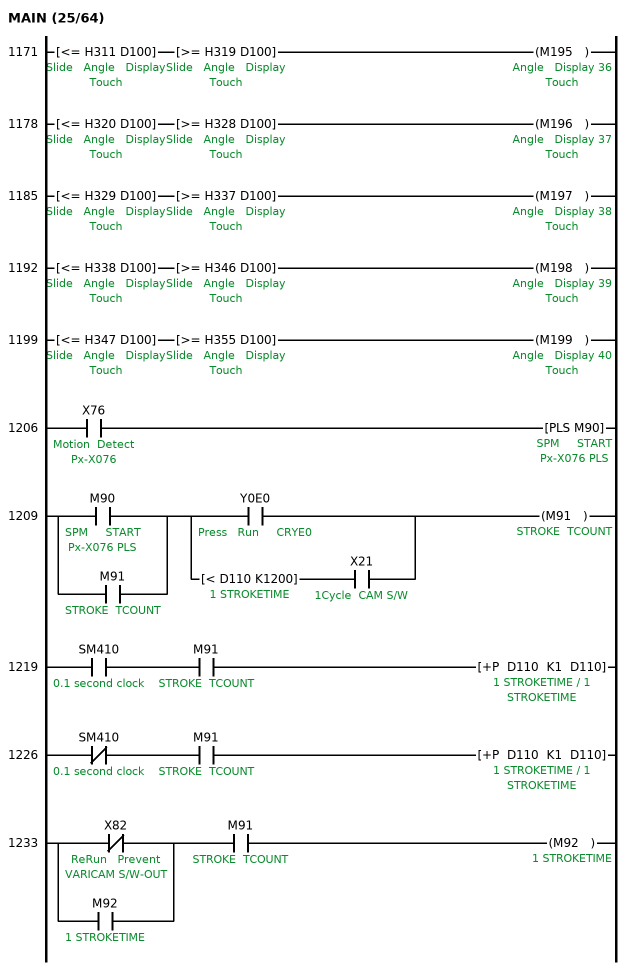
[picture p24: ladder of MAIN, rungs at steps 1171 to 1233]
1171  LD<=    H311 D100  ; Slide   Angle   Display Touch
      AND>=   H319 D100  ; Slide   Angle   Display Touch
      OUT     M195  ; Angle   Display 36      Touch
1178  LD<=    H320 D100  ; Slide   Angle   Display Touch
      AND>=   H328 D100  ; Slide   Angle   Display Touch
      OUT     M196  ; Angle   Display 37      Touch
1185  LD<=    H329 D100  ; Slide   Angle   Display Touch
      AND>=   H337 D100  ; Slide   Angle   Display Touch
      OUT     M197  ; Angle   Display 38      Touch
1192  LD<=    H338 D100  ; Slide   Angle   Display Touch
      AND>=   H346 D100  ; Slide   Angle   Display Touch
      OUT     M198  ; Angle   Display 39      Touch
1199  LD<=    H347 D100  ; Slide   Angle   Display Touch
      AND>=   H355 D100  ; Slide   Angle   Display Touch
      OUT     M199  ; Angle   Display 40      Touch
1206  LD      X76  ; Motion  Detect  Px-X076
      PLS     M90  ; SPM     START   Px-X076 PLS
1209  LD      M90  ; SPM     START   Px-X076 PLS
      OR      M91  ; STROKE  TCOUNT
      LD      Y0E0  ; Press   Run     CRYE0
      LD<     D110 K1200  ; 1 STROKETIME
      AND     X21  ; 1Cycle  CAM S/W
      ORB
      ANB
      OUT     M91  ; STROKE  TCOUNT
1219  LD      SM410  ; 0.1 second clock
      AND     M91  ; STROKE  TCOUNT
      +P      D110 K1 D110
1226  LDI     SM410  ; 0.1 second clock
      AND     M91  ; STROKE  TCOUNT
      +P      D110 K1 D110
1233  LDI     X82  ; ReRun   Prevent VARICAM S/W-OUT
      OR      M92  ; 1 STROKETIME
      AND     M91  ; STROKE  TCOUNT
      OUT     M92  ; 1 STROKETIME
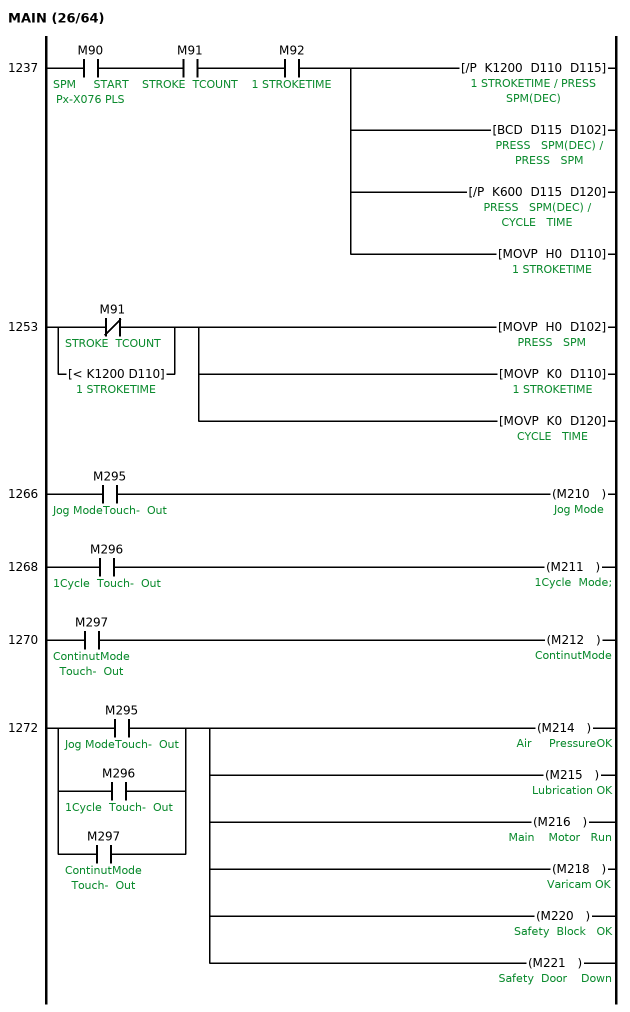
1237  LD      M90  ; SPM     START   Px-X076 PLS
      AND     M91  ; STROKE  TCOUNT
      AND     M92  ; 1 STROKETIME
      /P      K1200 D110 D115  ; PRESS   SPM(DEC)
      BCD     D115 D102  ; PRESS   SPM
      /P      K600 D115 D120  ; CYCLE   TIME
      MOVP    H0 D110
1253  LDI     M91  ; STROKE  TCOUNT
      OR<     K1200 D110  ; 1 STROKETIME
      MOVP    H0 D102
      MOVP    K0 D110
      MOVP    K0 D120
1266  LD      M295  ; Jog ModeTouch-  Out
      OUT     M210  ; Jog Mode
1268  LD      M296  ; 1Cycle  Touch-  Out
      OUT     M211  ; 1Cycle  Mode;
1270  LD      M297  ; ContinutMode    Touch-  Out
      OUT     M212  ; ContinutMode
1272  LD      M295  ; Jog ModeTouch-  Out
      OR      M296  ; 1Cycle  Touch-  Out
      OR      M297  ; ContinutMode    Touch-  Out
      OUT     M214  ; Air     PressureOK
      OUT     M215  ; Lubrication OK
      OUT     M216  ; Main    Motor   Run
      OUT     M218  ; Varicam OK
      OUT     M220  ; Safety  Block   OK
      OUT     M221  ; Safety  Door    Down
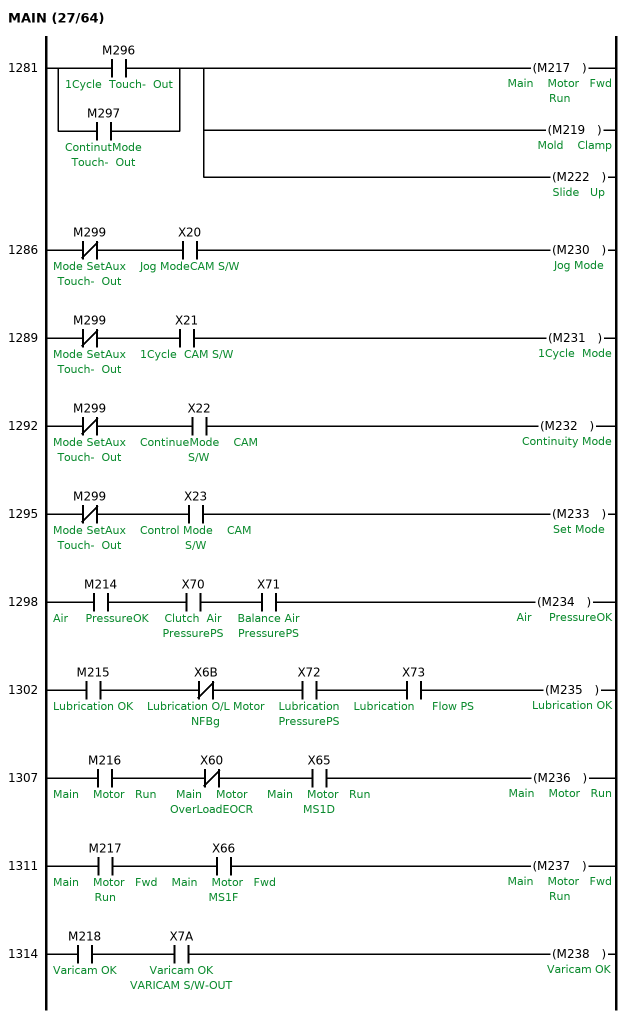
1281  LD      M296  ; 1Cycle  Touch-  Out
      OR      M297  ; ContinutMode    Touch-  Out
      OUT     M217  ; Main    Motor   Fwd Run
      OUT     M219  ; Mold    Clamp
      OUT     M222  ; Slide   Up
1286  LDI     M299  ; Mode SetAux     Touch-  Out
      AND     X20  ; Jog ModeCAM S/W
      OUT     M230  ; Jog Mode
1289  LDI     M299  ; Mode SetAux     Touch-  Out
      AND     X21  ; 1Cycle  CAM S/W
      OUT     M231  ; 1Cycle  Mode
1292  LDI     M299  ; Mode SetAux     Touch-  Out
      AND     X22  ; ContinueMode    CAM S/W
      OUT     M232  ; Continuity Mode
1295  LDI     M299  ; Mode SetAux     Touch-  Out
      AND     X23  ; Control Mode    CAM S/W
      OUT     M233  ; Set Mode
1298  LD      M214  ; Air     PressureOK
      AND     X70  ; Clutch  Air     PressurePS
      AND     X71  ; Balance Air     PressurePS
      OUT     M234  ; Air     PressureOK
1302  LD      M215  ; Lubrication OK
      ANI     X6B  ; Lubrication O/L Motor   NFBg
      AND     X72  ; Lubrication     PressurePS
      AND     X73  ; Lubrication     Flow PS
      OUT     M235  ; Lubrication OK
1307  LD      M216  ; Main    Motor   Run
      ANI     X60  ; Main    Motor   OverLoadEOCR
      AND     X65  ; Main    Motor   Run MS1D
      OUT     M236  ; Main    Motor   Run
1311  LD      M217  ; Main    Motor   Fwd Run
      AND     X66  ; Main    Motor   Fwd     MS1F
      OUT     M237  ; Main    Motor   Fwd Run
1314  LD      M218  ; Varicam OK
      AND     X7A  ; Varicam OK      VARICAM S/W-OUT
      OUT     M238  ; Varicam OK
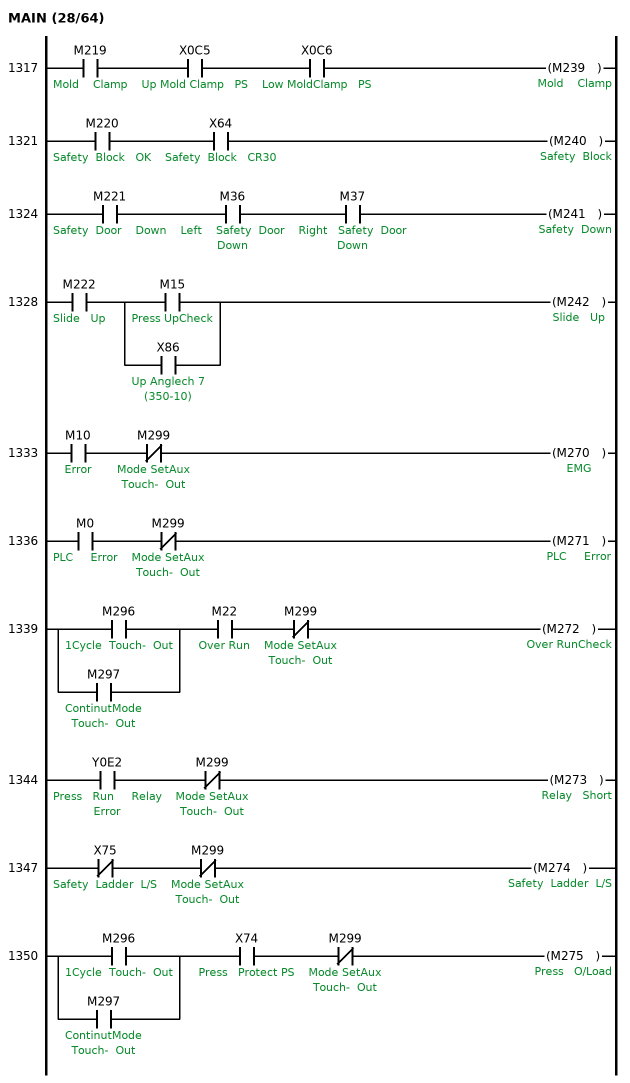
1317  LD      M219  ; Mold    Clamp
      AND     X0C5  ; Up Mold Clamp   PS
      AND     X0C6  ; Low MoldClamp   PS
      OUT     M239  ; Mold    Clamp
1321  LD      M220  ; Safety  Block   OK
      AND     X64  ; Safety  Block   CR30
      OUT     M240  ; Safety  Block
1324  LD      M221  ; Safety  Door    Down
      AND     M36  ; Left    Safety  Door    Down
      AND     M37  ; Right   Safety  Door    Down
      OUT     M241  ; Safety  Down
1328  LD      M222  ; Slide   Up
      LD      M15  ; Press UpCheck
      OR      X86  ; Up Anglech 7    (350-10)
      ANB
      OUT     M242  ; Slide   Up
1333  LD      M10  ; Error
      ANI     M299  ; Mode SetAux     Touch-  Out
      OUT     M270  ; EMG
1336  LD      M0  ; PLC     Error
      ANI     M299  ; Mode SetAux     Touch-  Out
      OUT     M271  ; PLC     Error
1339  LD      M296  ; 1Cycle  Touch-  Out
      OR      M297  ; ContinutMode    Touch-  Out
      AND     M22  ; Over Run
      ANI     M299  ; Mode SetAux     Touch-  Out
      OUT     M272  ; Over RunCheck
1344  LD      Y0E2  ; Press   Run     Relay   Error
      ANI     M299  ; Mode SetAux     Touch-  Out
      OUT     M273  ; Relay   Short
1347  LDI     X75  ; Safety  Ladder  L/S
      ANI     M299  ; Mode SetAux     Touch-  Out
      OUT     M274  ; Safety  Ladder  L/S
1350  LD      M296  ; 1Cycle  Touch-  Out
      OR      M297  ; ContinutMode    Touch-  Out
      AND     X74  ; Press   Protect PS
      ANI     M299  ; Mode SetAux     Touch-  Out
      OUT     M275  ; Press   O/Load
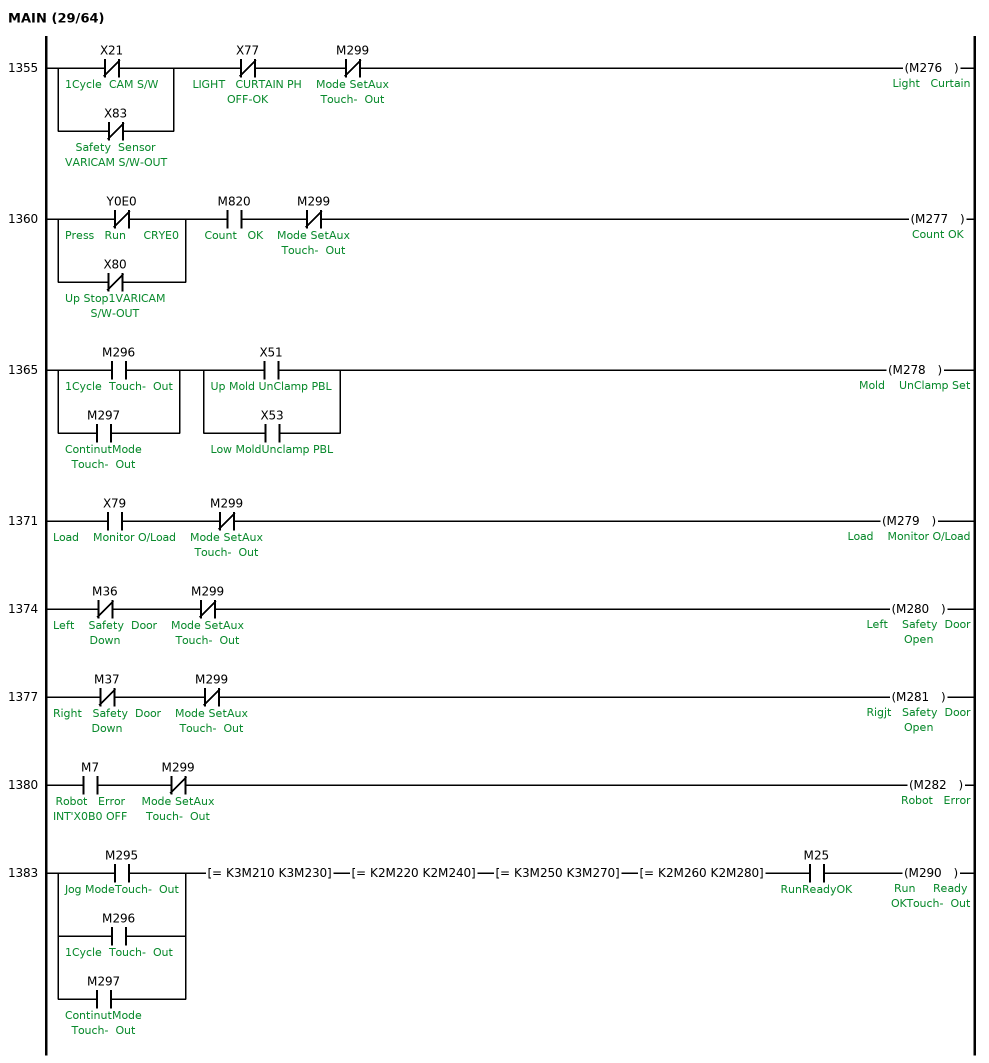
1355  LDI     X21  ; 1Cycle  CAM S/W
      ORI     X83  ; Safety  Sensor  VARICAM S/W-OUT
      ANI     X77  ; LIGHT   CURTAIN PH      OFF-OK
      ANI     M299  ; Mode SetAux     Touch-  Out
      OUT     M276  ; Light   Curtain
1360  LDI     Y0E0  ; Press   Run     CRYE0
      ORI     X80  ; Up Stop1VARICAM S/W-OUT
      AND     M820  ; Count   OK
      ANI     M299  ; Mode SetAux     Touch-  Out
      OUT     M277  ; Count OK
1365  LD      M296  ; 1Cycle  Touch-  Out
      OR      M297  ; ContinutMode    Touch-  Out
      LD      X51  ; Up Mold UnClamp PBL
      OR      X53  ; Low MoldUnclamp PBL
      ANB
      OUT     M278  ; Mold    UnClamp Set
1371  LD      X79  ; Load    Monitor O/Load
      ANI     M299  ; Mode SetAux     Touch-  Out
      OUT     M279  ; Load    Monitor O/Load
1374  LDI     M36  ; Left    Safety  Door    Down
      ANI     M299  ; Mode SetAux     Touch-  Out
      OUT     M280  ; Left    Safety  Door    Open
1377  LDI     M37  ; Right   Safety  Door    Down
      ANI     M299  ; Mode SetAux     Touch-  Out
      OUT     M281  ; Rigjt   Safety  Door    Open
1380  LD      M7  ; Robot   Error   INT'X0B0 OFF
      ANI     M299  ; Mode SetAux     Touch-  Out
      OUT     M282  ; Robot   Error
1383  LD      M295  ; Jog ModeTouch-  Out
      OR      M296  ; 1Cycle  Touch-  Out
      OR      M297  ; ContinutMode    Touch-  Out
      AND=    K3M210 K3M230  ; Jog Mode / Jog Mode
      AND=    K2M220 K2M240  ; Safety  Block   OK / Safety  Block
      AND=    K3M250 K3M270  ; EMG / EMG
      AND=    K2M260 K2M280  ; Left    Safety  Door    Open / Left    Safety  Door    Open
      AND     M25  ; RunReadyOK
      OUT     M290  ; Run     Ready OKTouch-  Out
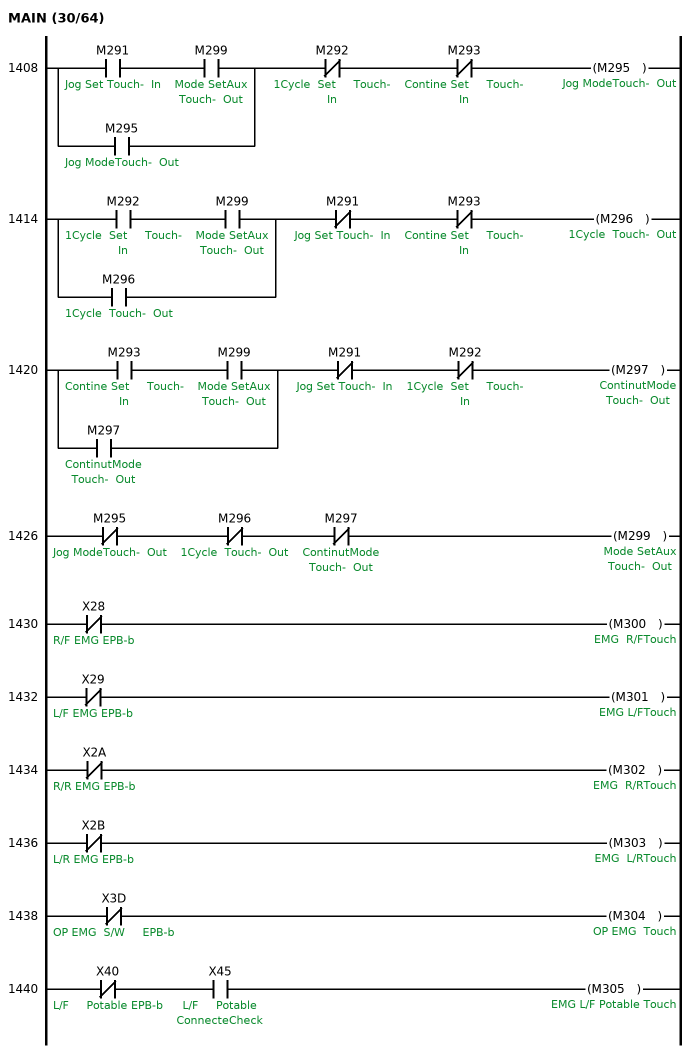
1408  LD      M291  ; Jog Set Touch-  In
      AND     M299  ; Mode SetAux     Touch-  Out
      OR      M295  ; Jog ModeTouch-  Out
      ANI     M292  ; 1Cycle  Set     Touch-  In
      ANI     M293  ; Contine Set     Touch-  In
      OUT     M295  ; Jog ModeTouch-  Out
1414  LD      M292  ; 1Cycle  Set     Touch-  In
      AND     M299  ; Mode SetAux     Touch-  Out
      OR      M296  ; 1Cycle  Touch-  Out
      ANI     M291  ; Jog Set Touch-  In
      ANI     M293  ; Contine Set     Touch-  In
      OUT     M296  ; 1Cycle  Touch-  Out
1420  LD      M293  ; Contine Set     Touch-  In
      AND     M299  ; Mode SetAux     Touch-  Out
      OR      M297  ; ContinutMode    Touch-  Out
      ANI     M291  ; Jog Set Touch-  In
      ANI     M292  ; 1Cycle  Set     Touch-  In
      OUT     M297  ; ContinutMode    Touch-  Out
1426  LDI     M295  ; Jog ModeTouch-  Out
      ANI     M296  ; 1Cycle  Touch-  Out
      ANI     M297  ; ContinutMode    Touch-  Out
      OUT     M299  ; Mode SetAux     Touch-  Out
1430  LDI     X28  ; R/F EMG EPB-b
      OUT     M300  ; EMG  R/FTouch
1432  LDI     X29  ; L/F EMG EPB-b
      OUT     M301  ; EMG L/FTouch
1434  LDI     X2A  ; R/R EMG EPB-b
      OUT     M302  ; EMG  R/RTouch
1436  LDI     X2B  ; L/R EMG EPB-b
      OUT     M303  ; EMG  L/RTouch
1438  LDI     X3D  ; OP EMG  S/W     EPB-b
      OUT     M304  ; OP EMG  Touch
1440  LDI     X40  ; L/F     Potable EPB-b
      AND     X45  ; L/F     Potable ConnecteCheck
      OUT     M305  ; EMG L/F Potable Touch
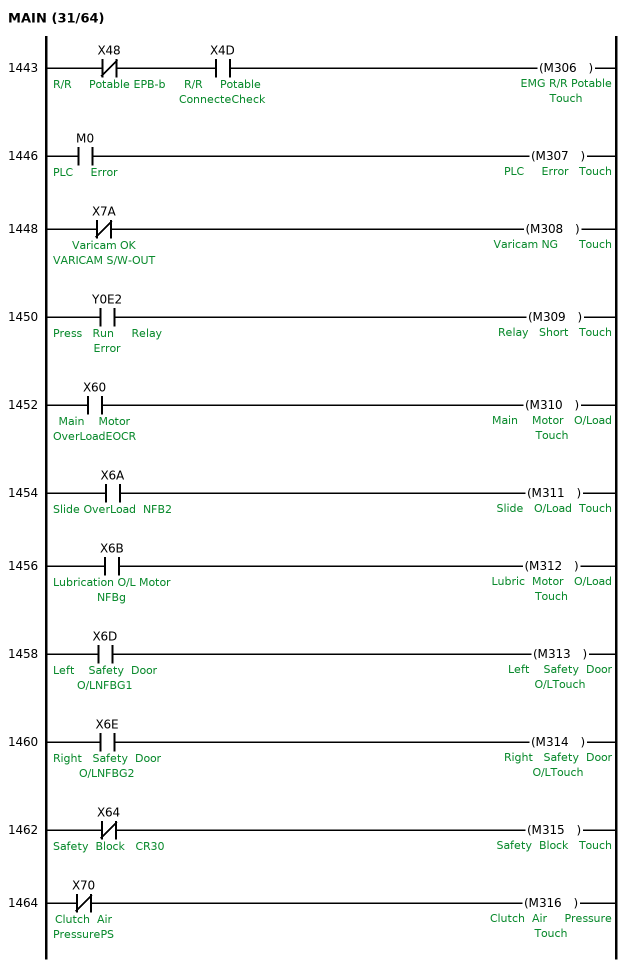
1443  LDI     X48  ; R/R     Potable EPB-b
      AND     X4D  ; R/R     Potable ConnecteCheck
      OUT     M306  ; EMG R/R Potable Touch
1446  LD      M0  ; PLC     Error
      OUT     M307  ; PLC     Error   Touch
1448  LDI     X7A  ; Varicam OK      VARICAM S/W-OUT
      OUT     M308  ; Varicam NG      Touch
1450  LD      Y0E2  ; Press   Run     Relay   Error
      OUT     M309  ; Relay   Short   Touch
1452  LD      X60  ; Main    Motor   OverLoadEOCR
      OUT     M310  ; Main    Motor   O/Load  Touch
1454  LD      X6A  ; Slide OverLoad  NFB2
      OUT     M311  ; Slide   O/Load  Touch
1456  LD      X6B  ; Lubrication O/L Motor   NFBg
      OUT     M312  ; Lubric  Motor   O/Load  Touch
1458  LD      X6D  ; Left    Safety  Door O/LNFBG1
      OUT     M313  ; Left    Safety  Door O/LTouch
1460  LD      X6E  ; Right   Safety  Door O/LNFBG2
      OUT     M314  ; Right   Safety  Door O/LTouch
1462  LDI     X64  ; Safety  Block   CR30
      OUT     M315  ; Safety  Block   Touch
1464  LDI     X70  ; Clutch  Air     PressurePS
      OUT     M316  ; Clutch  Air     Pressure Touch
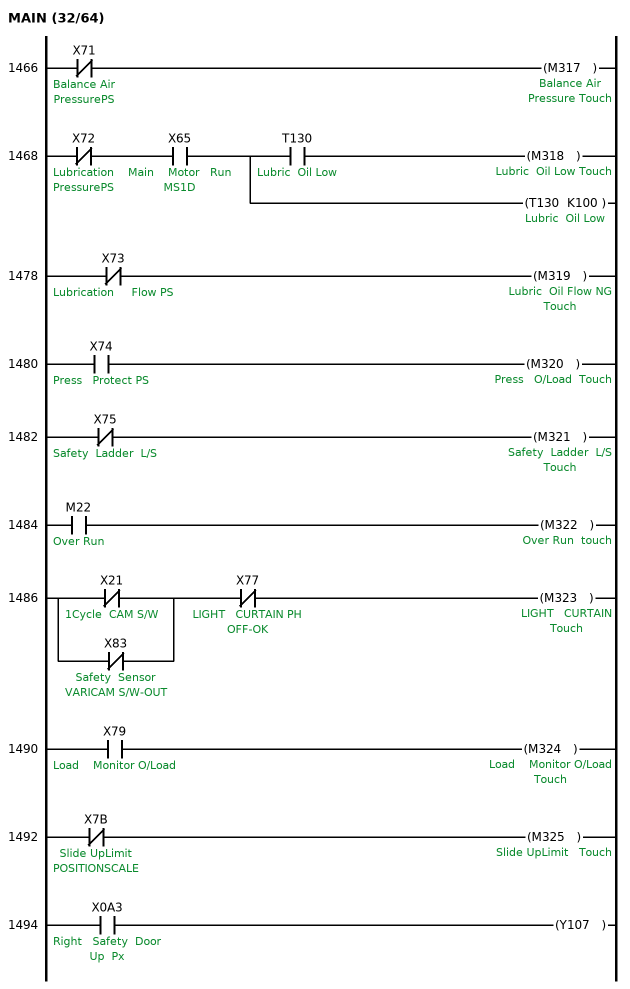
1466  LDI     X71  ; Balance Air     PressurePS
      OUT     M317  ; Balance Air     Pressure Touch
1468  LDI     X72  ; Lubrication     PressurePS
      AND     X65  ; Main    Motor   Run MS1D
      MPS
      AND     T130  ; Lubric  Oil Low
      OUT     M318  ; Lubric  Oil Low Touch
      MPP
      OUT     T130 K100  ; Lubric  Oil Low
1478  LDI     X73  ; Lubrication     Flow PS
      OUT     M319  ; Lubric  Oil Flow NG     Touch
1480  LD      X74  ; Press   Protect PS
      OUT     M320  ; Press   O/Load  Touch
1482  LDI     X75  ; Safety  Ladder  L/S
      OUT     M321  ; Safety  Ladder  L/S     Touch
1484  LD      M22  ; Over Run
      OUT     M322  ; Over Run  touch
1486  LDI     X21  ; 1Cycle  CAM S/W
      ORI     X83  ; Safety  Sensor  VARICAM S/W-OUT
      ANI     X77  ; LIGHT   CURTAIN PH      OFF-OK
      OUT     M323  ; LIGHT   CURTAIN Touch
1490  LD      X79  ; Load    Monitor O/Load
      OUT     M324  ; Load    Monitor O/Load  Touch
1492  LDI     X7B  ; Slide UpLimit   POSITIONSCALE
      OUT     M325  ; Slide UpLimit   Touch
1494  LD      X0A3  ; Right   Safety  Door Up  Px
      OUT     Y107
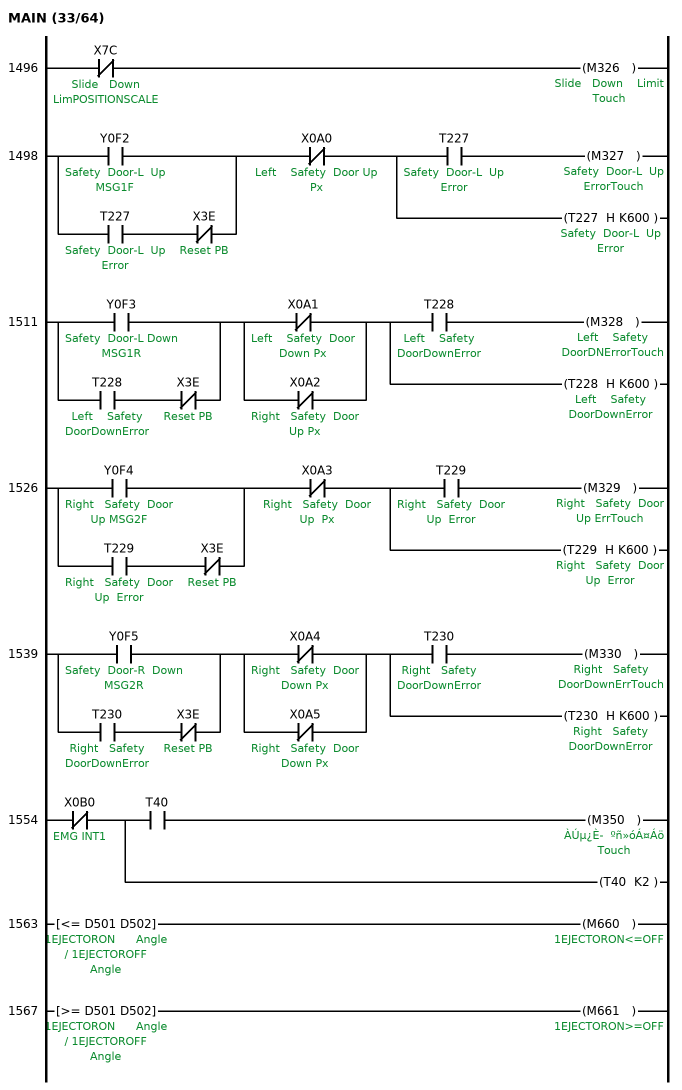
1496  LDI     X7C  ; Slide   Down LimPOSITIONSCALE
      OUT     M326  ; Slide   Down    Limit   Touch
1498  LD      Y0F2  ; Safety  Door-L  Up MSG1F
      LD      T227  ; Safety  Door-L  Up Error
      ANI     X3E  ; Reset PB
      ORB
      ANI     X0A0  ; Left    Safety  Door Up Px
      MPS
      AND     T227  ; Safety  Door-L  Up Error
      OUT     M327  ; Safety  Door-L  Up ErrorTouch
      MPP
      OUTH    T227 K600  ; Safety  Door-L  Up Error
1511  LD      Y0F3  ; Safety  Door-L Down     MSG1R
      LD      T228  ; Left    Safety  DoorDownError
      ANI     X3E  ; Reset PB
      ORB
      LDI     X0A1  ; Left    Safety  Door    Down Px
      ORI     X0A2  ; Right   Safety  Door Up Px
      ANB
      MPS
      AND     T228  ; Left    Safety  DoorDownError
      OUT     M328  ; Left    Safety  DoorDNErrorTouch
      MPP
      OUTH    T228 K600  ; Left    Safety  DoorDownError
1526  LD      Y0F4  ; Right   Safety  Door Up MSG2F
      LD      T229  ; Right   Safety  Door Up  Error
      ANI     X3E  ; Reset PB
      ORB
      ANI     X0A3  ; Right   Safety  Door Up  Px
      MPS
      AND     T229  ; Right   Safety  Door Up  Error
      OUT     M329  ; Right   Safety  Door Up ErrTouch
      MPP
      OUTH    T229 K600  ; Right   Safety  Door Up  Error
1539  LD      Y0F5  ; Safety  Door-R  Down    MSG2R
      LD      T230  ; Right   Safety  DoorDownError
      ANI     X3E  ; Reset PB
      ORB
      LDI     X0A4  ; Right   Safety  Door    Down Px
      ORI     X0A5  ; Right   Safety  Door    Down Px
      ANB
      MPS
      AND     T230  ; Right   Safety  DoorDownError
      OUT     M330  ; Right   Safety  DoorDownErrTouch
      MPP
      OUTH    T230 K600  ; Right   Safety  DoorDownError
1554  LDI     X0B0  ; EMG INT1
      MPS
      AND     T40
      OUT     M350  ; ÀÚµ¿È­  ºñ»óÁ¤ÁöTouch
      MPP
      OUT     T40 K2
1563  LD<=    D501 D502  ; 1EJECTORON      Angle / 1EJECTOROFF     Angle
      OUT     M660  ; 1EJECTORON<=OFF
1567  LD>=    D501 D502  ; 1EJECTORON      Angle / 1EJECTOROFF     Angle
      OUT     M661  ; 1EJECTORON>=OFF
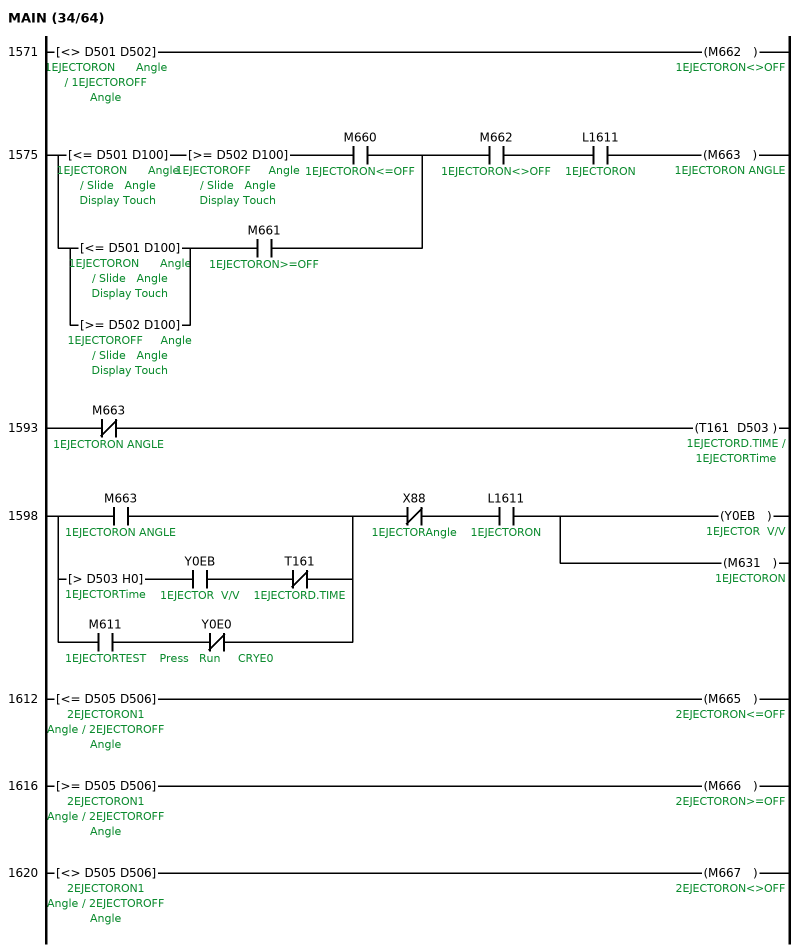
1571  LD<>    D501 D502  ; 1EJECTORON      Angle / 1EJECTOROFF     Angle
      OUT     M662  ; 1EJECTORON<>OFF
1575  LD<=    D501 D100  ; 1EJECTORON      Angle / Slide   Angle   Display Touch
      AND>=   D502 D100  ; 1EJECTOROFF     Angle / Slide   Angle   Display Touch
      AND     M660  ; 1EJECTORON<=OFF
      LD<=    D501 D100  ; 1EJECTORON      Angle / Slide   Angle   Display Touch
      OR>=    D502 D100  ; 1EJECTOROFF     Angle / Slide   Angle   Display Touch
      AND     M661  ; 1EJECTORON>=OFF
      ORB
      AND     M662  ; 1EJECTORON<>OFF
      AND     L1611  ; 1EJECTORON
      OUT     M663  ; 1EJECTORON ANGLE
1593  LDI     M663  ; 1EJECTORON ANGLE
      OUT     T161 D503  ; 1EJECTORD.TIME / 1EJECTORTime
1598  LD      M663  ; 1EJECTORON ANGLE
      LD>     D503 H0  ; 1EJECTORTime
      AND     Y0EB  ; 1EJECTOR  V/V
      ANI     T161  ; 1EJECTORD.TIME
      ORB
      LD      M611  ; 1EJECTORTEST
      ANI     Y0E0  ; Press   Run     CRYE0
      ORB
      ANI     X88  ; 1EJECTORAngle
      AND     L1611  ; 1EJECTORON
      OUT     Y0EB  ; 1EJECTOR  V/V
      OUT     M631  ; 1EJECTORON
1612  LD<=    D505 D506  ; 2EJECTORON1     Angle / 2EJECTOROFF     Angle
      OUT     M665  ; 2EJECTORON<=OFF
1616  LD>=    D505 D506  ; 2EJECTORON1     Angle / 2EJECTOROFF     Angle
      OUT     M666  ; 2EJECTORON>=OFF
1620  LD<>    D505 D506  ; 2EJECTORON1     Angle / 2EJECTOROFF     Angle
      OUT     M667  ; 2EJECTORON<>OFF
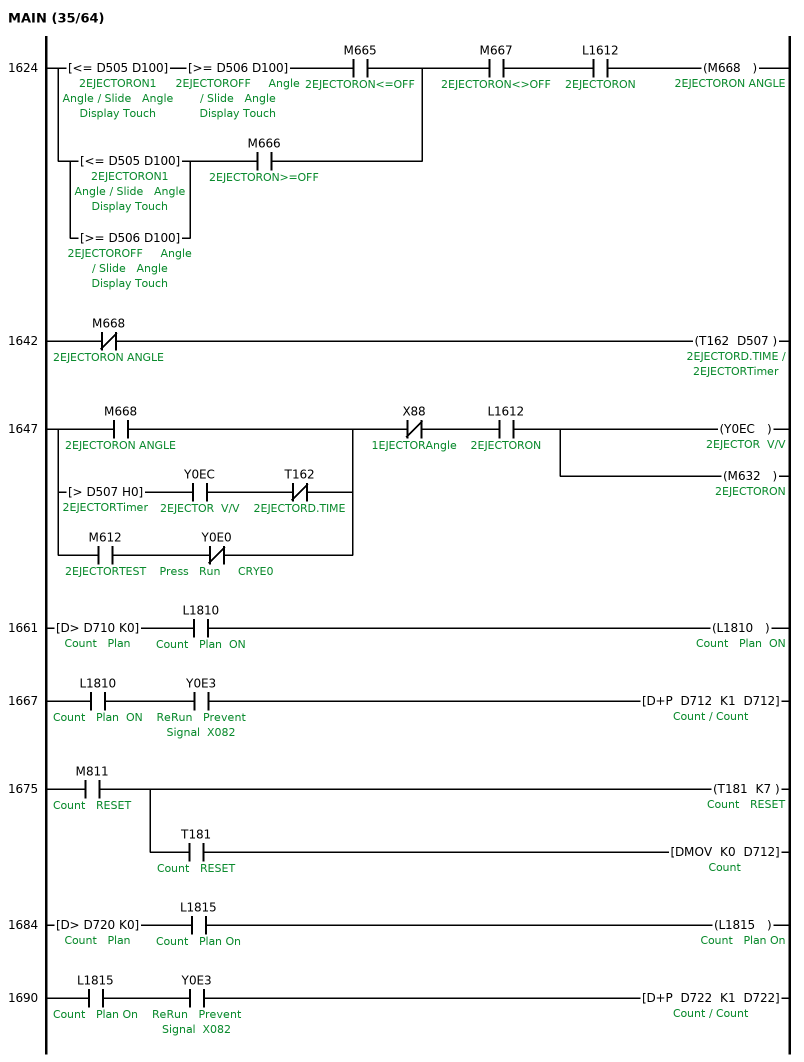
1624  LD<=    D505 D100  ; 2EJECTORON1     Angle / Slide   Angle   Display Touch
      AND>=   D506 D100  ; 2EJECTOROFF     Angle / Slide   Angle   Display Touch
      AND     M665  ; 2EJECTORON<=OFF
      LD<=    D505 D100  ; 2EJECTORON1     Angle / Slide   Angle   Display Touch
      OR>=    D506 D100  ; 2EJECTOROFF     Angle / Slide   Angle   Display Touch
      AND     M666  ; 2EJECTORON>=OFF
      ORB
      AND     M667  ; 2EJECTORON<>OFF
      AND     L1612  ; 2EJECTORON
      OUT     M668  ; 2EJECTORON ANGLE
1642  LDI     M668  ; 2EJECTORON ANGLE
      OUT     T162 D507  ; 2EJECTORD.TIME / 2EJECTORTimer
1647  LD      M668  ; 2EJECTORON ANGLE
      LD>     D507 H0  ; 2EJECTORTimer
      AND     Y0EC  ; 2EJECTOR  V/V
      ANI     T162  ; 2EJECTORD.TIME
      ORB
      LD      M612  ; 2EJECTORTEST
      ANI     Y0E0  ; Press   Run     CRYE0
      ORB
      ANI     X88  ; 1EJECTORAngle
      AND     L1612  ; 2EJECTORON
      OUT     Y0EC  ; 2EJECTOR  V/V
      OUT     M632  ; 2EJECTORON
1661  LDD>    D710 K0  ; Count   Plan
      AND     L1810  ; Count   Plan  ON
      OUT     L1810  ; Count   Plan  ON
1667  LD      L1810  ; Count   Plan  ON
      AND     Y0E3  ; ReRun   Prevent Signal  X082
      D+P     D712 K1 D712  ; Count
1675  LD      M811  ; Count   RESET
      OUT     T181 K7  ; Count   RESET
      AND     T181  ; Count   RESET
      DMOV    K0 D712
1684  LDD>    D720 K0  ; Count   Plan
      AND     L1815  ; Count   Plan On
      OUT     L1815  ; Count   Plan On
1690  LD      L1815  ; Count   Plan On
      AND     Y0E3  ; ReRun   Prevent Signal  X082
      D+P     D722 K1 D722  ; Count
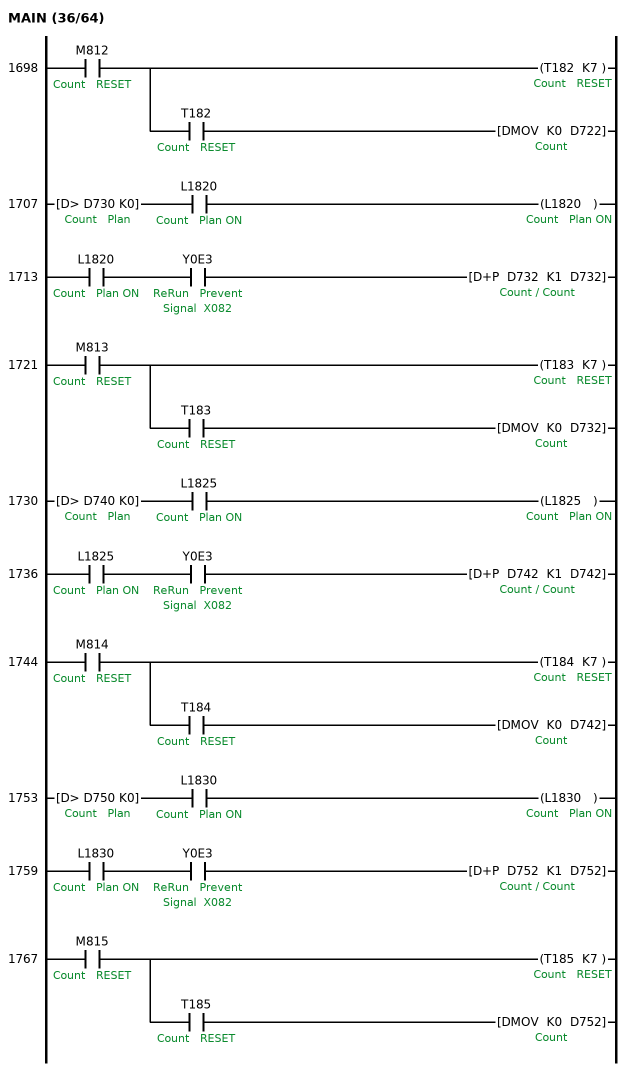
1698  LD      M812  ; Count   RESET
      OUT     T182 K7  ; Count   RESET
      AND     T182  ; Count   RESET
      DMOV    K0 D722
1707  LDD>    D730 K0  ; Count   Plan
      AND     L1820  ; Count   Plan ON
      OUT     L1820  ; Count   Plan ON
1713  LD      L1820  ; Count   Plan ON
      AND     Y0E3  ; ReRun   Prevent Signal  X082
      D+P     D732 K1 D732  ; Count
1721  LD      M813  ; Count   RESET
      OUT     T183 K7  ; Count   RESET
      AND     T183  ; Count   RESET
      DMOV    K0 D732
1730  LDD>    D740 K0  ; Count   Plan
      AND     L1825  ; Count   Plan ON
      OUT     L1825  ; Count   Plan ON
1736  LD      L1825  ; Count   Plan ON
      AND     Y0E3  ; ReRun   Prevent Signal  X082
      D+P     D742 K1 D742  ; Count
1744  LD      M814  ; Count   RESET
      OUT     T184 K7  ; Count   RESET
      AND     T184  ; Count   RESET
      DMOV    K0 D742
1753  LDD>    D750 K0  ; Count   Plan
      AND     L1830  ; Count   Plan ON
      OUT     L1830  ; Count   Plan ON
1759  LD      L1830  ; Count   Plan ON
      AND     Y0E3  ; ReRun   Prevent Signal  X082
      D+P     D752 K1 D752  ; Count
1767  LD      M815  ; Count   RESET
      OUT     T185 K7  ; Count   RESET
      AND     T185  ; Count   RESET
      DMOV    K0 D752
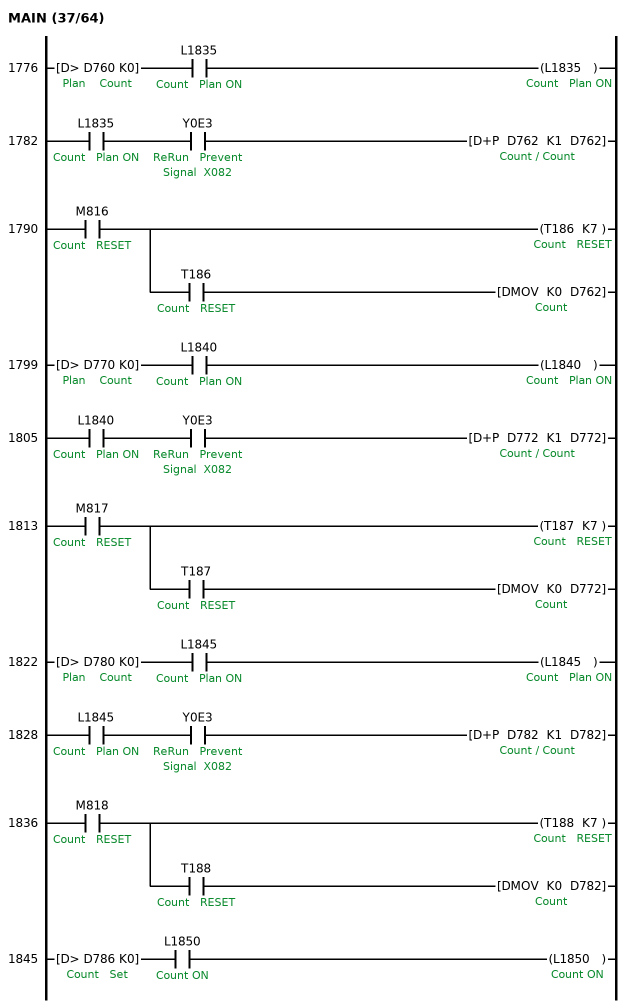
1776  LDD>    D760 K0  ; Plan    Count
      AND     L1835  ; Count   Plan ON
      OUT     L1835  ; Count   Plan ON
1782  LD      L1835  ; Count   Plan ON
      AND     Y0E3  ; ReRun   Prevent Signal  X082
      D+P     D762 K1 D762  ; Count
1790  LD      M816  ; Count   RESET
      OUT     T186 K7  ; Count   RESET
      AND     T186  ; Count   RESET
      DMOV    K0 D762
1799  LDD>    D770 K0  ; Plan    Count
      AND     L1840  ; Count   Plan ON
      OUT     L1840  ; Count   Plan ON
1805  LD      L1840  ; Count   Plan ON
      AND     Y0E3  ; ReRun   Prevent Signal  X082
      D+P     D772 K1 D772  ; Count
1813  LD      M817  ; Count   RESET
      OUT     T187 K7  ; Count   RESET
      AND     T187  ; Count   RESET
      DMOV    K0 D772
1822  LDD>    D780 K0  ; Plan    Count
      AND     L1845  ; Count   Plan ON
      OUT     L1845  ; Count   Plan ON
1828  LD      L1845  ; Count   Plan ON
      AND     Y0E3  ; ReRun   Prevent Signal  X082
      D+P     D782 K1 D782  ; Count
1836  LD      M818  ; Count   RESET
      OUT     T188 K7  ; Count   RESET
      AND     T188  ; Count   RESET
      DMOV    K0 D782
1845  LDD>    D786 K0  ; Count   Set
      AND     L1850  ; Count ON
      OUT     L1850  ; Count ON
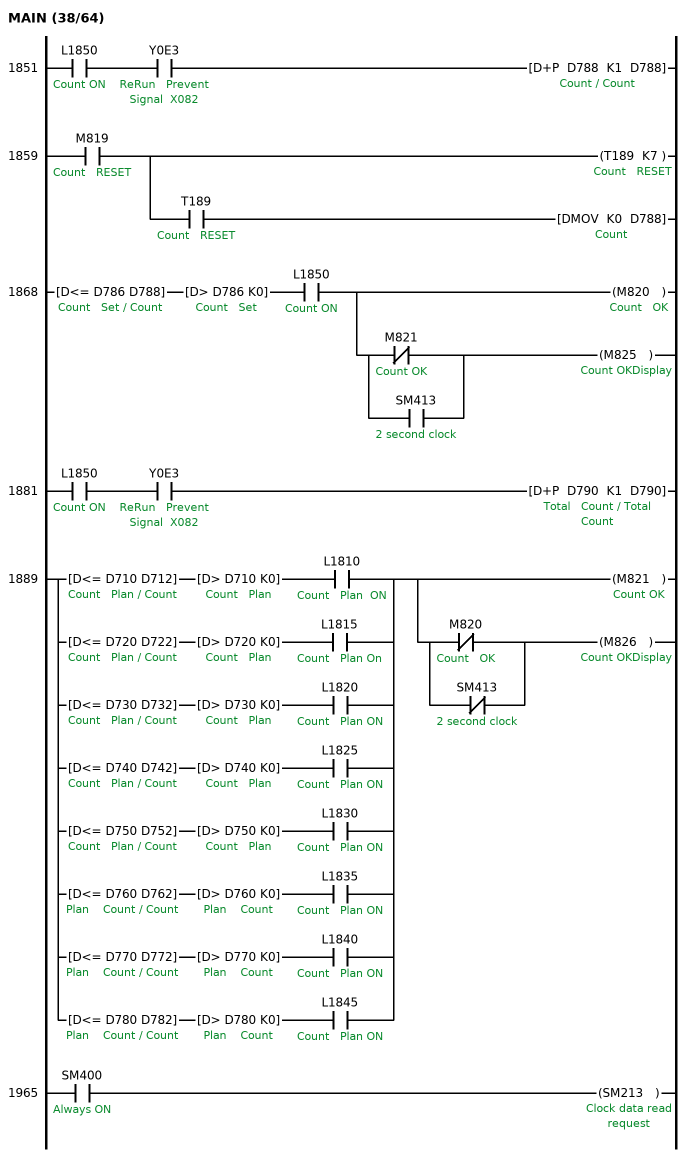
1851  LD      L1850  ; Count ON
      AND     Y0E3  ; ReRun   Prevent Signal  X082
      D+P     D788 K1 D788  ; Count
1859  LD      M819  ; Count   RESET
      OUT     T189 K7  ; Count   RESET
      AND     T189  ; Count   RESET
      DMOV    K0 D788
1868  LDD<=   D786 D788  ; Count   Set / Count
      ANDD>   D786 K0  ; Count   Set
      AND     L1850  ; Count ON
      OUT     M820  ; Count   OK
      LDI     M821  ; Count OK
      OR      SM413  ; 2 second clock
      ANB
      OUT     M825  ; Count OKDisplay
1881  LD      L1850  ; Count ON
      AND     Y0E3  ; ReRun   Prevent Signal  X082
      D+P     D790 K1 D790  ; Total   Count
1889  LDD<=   D710 D712  ; Count   Plan / Count
      ANDD>   D710 K0  ; Count   Plan
      AND     L1810  ; Count   Plan  ON
      LDD<=   D720 D722  ; Count   Plan / Count
      ANDD>   D720 K0  ; Count   Plan
      AND     L1815  ; Count   Plan On
      ORB
      LDD<=   D730 D732  ; Count   Plan / Count
      ANDD>   D730 K0  ; Count   Plan
      AND     L1820  ; Count   Plan ON
      ORB
      LDD<=   D740 D742  ; Count   Plan / Count
      ANDD>   D740 K0  ; Count   Plan
      AND     L1825  ; Count   Plan ON
      ORB
      LDD<=   D750 D752  ; Count   Plan / Count
      ANDD>   D750 K0  ; Count   Plan
      AND     L1830  ; Count   Plan ON
      ORB
      LDD<=   D760 D762  ; Plan    Count / Count
      ANDD>   D760 K0  ; Plan    Count
      AND     L1835  ; Count   Plan ON
      ORB
      LDD<=   D770 D772  ; Plan    Count / Count
      ANDD>   D770 K0  ; Plan    Count
      AND     L1840  ; Count   Plan ON
      ORB
      LDD<=   D780 D782  ; Plan    Count / Count
      ANDD>   D780 K0  ; Plan    Count
      AND     L1845  ; Count   Plan ON
      ORB
      OUT     M821  ; Count OK
      LDI     M820  ; Count   OK
      ORI     SM413  ; 2 second clock
      ANB
      OUT     M826  ; Count OKDisplay
1965  LD      SM400  ; Always ON
      OUT     SM213  ; Clock data read request
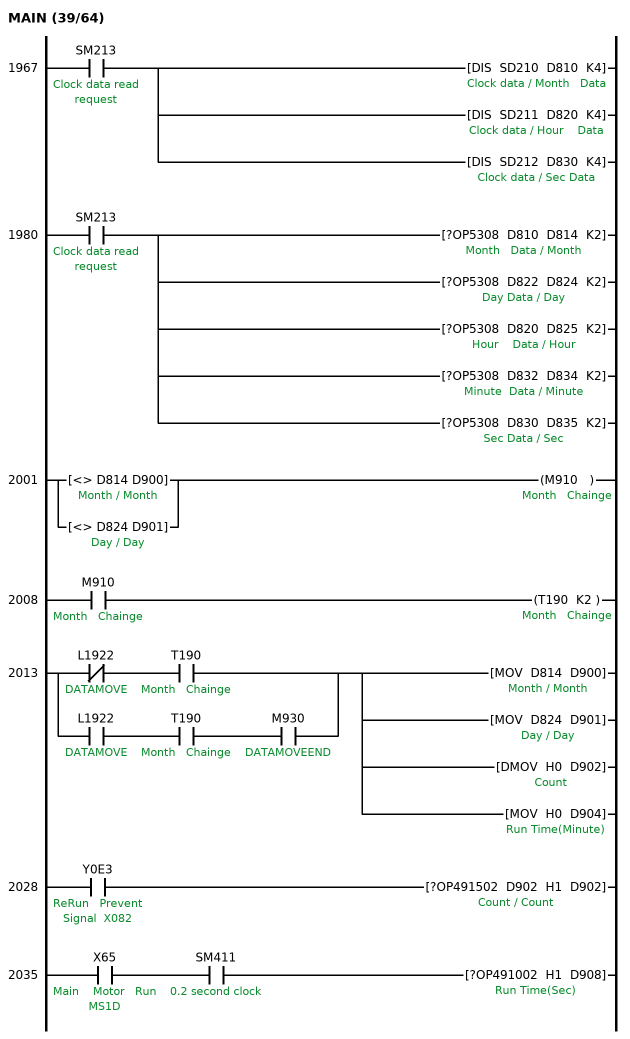
1967  LD      SM213  ; Clock data read request
      DIS     SD210 D810 K4  ; Clock data / Month   Data
      DIS     SD211 D820 K4  ; Clock data / Hour    Data
      DIS     SD212 D830 K4  ; Clock data / Sec Data
1980  LD      SM213  ; Clock data read request
      ?OP5308 D810 D814 K2  ; Month
      ?OP5308 D822 D824 K2  ; Day Data / Day
      ?OP5308 D820 D825 K2  ; Hour
      ?OP5308 D832 D834 K2  ; Minute  Data / Minute
      ?OP5308 D830 D835 K2  ; Sec
2001  LD<>    D814 D900  ; Month / Month
      OR<>    D824 D901  ; Day / Day
      OUT     M910  ; Month   Chainge
2008  LD      M910  ; Month   Chainge
      OUT     T190 K2  ; Month   Chainge
2013  LDI     L1922  ; DATAMOVE
      AND     T190  ; Month   Chainge
      LD      L1922  ; DATAMOVE
      AND     T190  ; Month   Chainge
      AND     M930  ; DATAMOVEEND
      ORB
      MOV     D814 D900
      MOV     D824 D901
      DMOV    H0 D902  ; Count
      MOV     H0 D904  ; Run Time(Minute)
2028  LD      Y0E3  ; ReRun   Prevent Signal  X082
      ?OP491502 D902 H1 D902
2035  LD      X65  ; Main    Motor   Run MS1D
      AND     SM411  ; 0.2 second clock
      ?OP491002 H1 D908  ; Run Time(Sec)
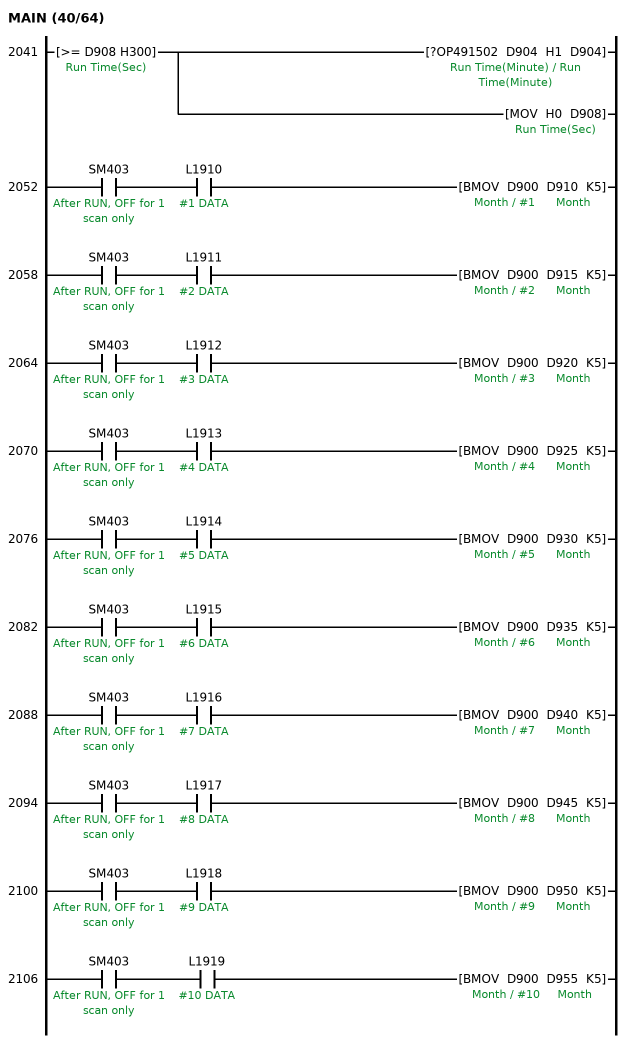
2041  LD>=    D908 H300  ; Run Time(Sec)
      ?OP491502 D904 H1 D904
      MOV     H0 D908
2052  LD      SM403  ; After RUN, OFF for 1 scan only
      AND     L1910  ; #1 DATA
      BMOV    D900 D910 K5  ; #1      Month
2058  LD      SM403  ; After RUN, OFF for 1 scan only
      AND     L1911  ; #2 DATA
      BMOV    D900 D915 K5  ; #2      Month
2064  LD      SM403  ; After RUN, OFF for 1 scan only
      AND     L1912  ; #3 DATA
      BMOV    D900 D920 K5  ; #3      Month
2070  LD      SM403  ; After RUN, OFF for 1 scan only
      AND     L1913  ; #4 DATA
      BMOV    D900 D925 K5  ; #4      Month
2076  LD      SM403  ; After RUN, OFF for 1 scan only
      AND     L1914  ; #5 DATA
      BMOV    D900 D930 K5  ; #5      Month
2082  LD      SM403  ; After RUN, OFF for 1 scan only
      AND     L1915  ; #6 DATA
      BMOV    D900 D935 K5  ; #6      Month
2088  LD      SM403  ; After RUN, OFF for 1 scan only
      AND     L1916  ; #7 DATA
      BMOV    D900 D940 K5  ; #7      Month
2094  LD      SM403  ; After RUN, OFF for 1 scan only
      AND     L1917  ; #8 DATA
      BMOV    D900 D945 K5  ; #8      Month
2100  LD      SM403  ; After RUN, OFF for 1 scan only
      AND     L1918  ; #9 DATA
      BMOV    D900 D950 K5  ; #9      Month
2106  LD      SM403  ; After RUN, OFF for 1 scan only
      AND     L1919  ; #10 DATA
      BMOV    D900 D955 K5  ; #10     Month
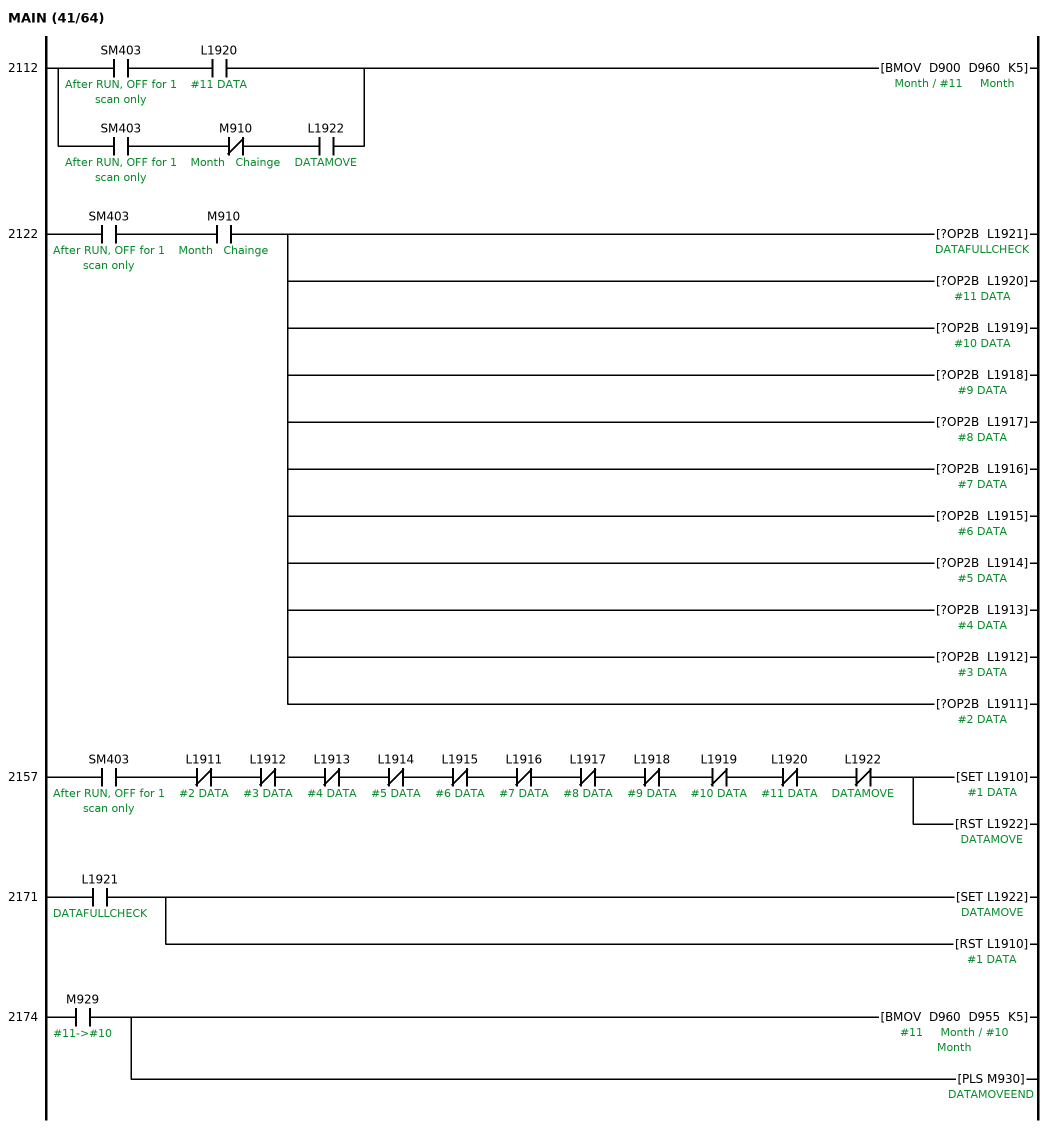
2112  LD      SM403  ; After RUN, OFF for 1 scan only
      AND     L1920  ; #11 DATA
      LD      SM403  ; After RUN, OFF for 1 scan only
      ANI     M910  ; Month   Chainge
      AND     L1922  ; DATAMOVE
      ORB
      BMOV    D900 D960 K5  ; #11     Month
2122  LD      SM403  ; After RUN, OFF for 1 scan only
      AND     M910  ; Month   Chainge
      ?OP2B   L1921  ; DATAFULLCHECK
      ?OP2B   L1920
      ?OP2B   L1919
      ?OP2B   L1918
      ?OP2B   L1917
      ?OP2B   L1916
      ?OP2B   L1915
      ?OP2B   L1914
      ?OP2B   L1913
      ?OP2B   L1912
      ?OP2B   L1911
2157  LD      SM403  ; After RUN, OFF for 1 scan only
      ANI     L1911  ; #2 DATA
      ANI     L1912  ; #3 DATA
      ANI     L1913  ; #4 DATA
      ANI     L1914  ; #5 DATA
      ANI     L1915  ; #6 DATA
      ANI     L1916  ; #7 DATA
      ANI     L1917  ; #8 DATA
      ANI     L1918  ; #9 DATA
      ANI     L1919  ; #10 DATA
      ANI     L1920  ; #11 DATA
      ANI     L1922  ; DATAMOVE
      SET     L1910  ; #1 DATA
      RST     L1922  ; DATAMOVE
2171  LD      L1921  ; DATAFULLCHECK
      SET     L1922  ; DATAMOVE
      RST     L1910  ; #1 DATA
2174  LD      M929  ; #11->#10
      BMOV    D960 D955 K5
      PLS     M930  ; DATAMOVEEND
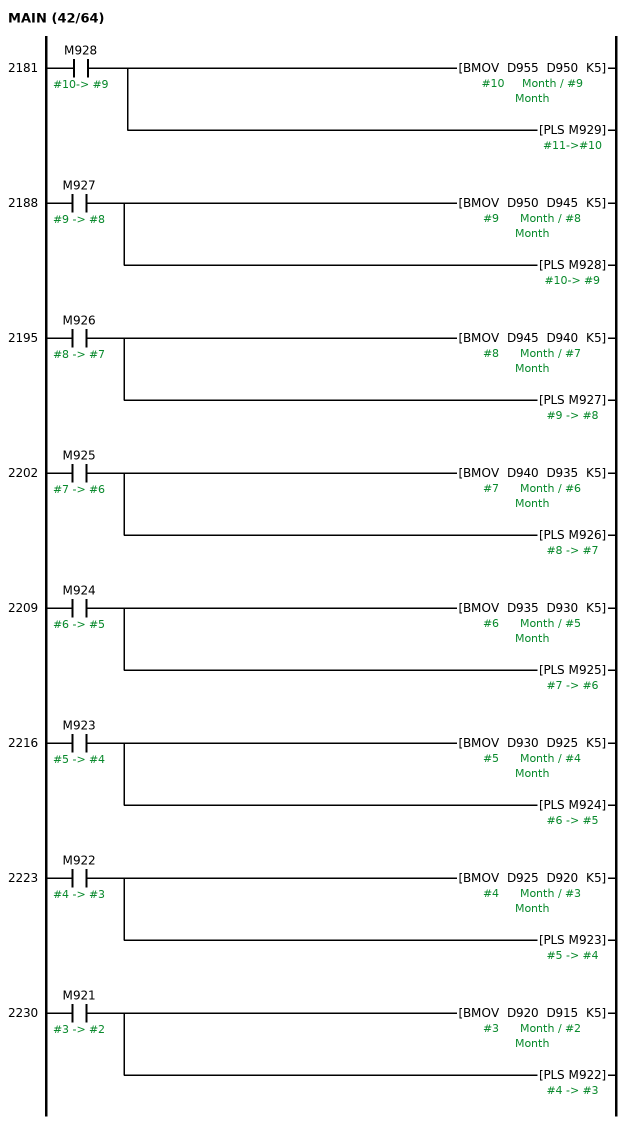
2181  LD      M928  ; #10-> #9
      BMOV    D955 D950 K5
      PLS     M929  ; #11->#10
2188  LD      M927  ; #9 -> #8
      BMOV    D950 D945 K5
      PLS     M928  ; #10-> #9
2195  LD      M926  ; #8 -> #7
      BMOV    D945 D940 K5
      PLS     M927  ; #9 -> #8
2202  LD      M925  ; #7 -> #6
      BMOV    D940 D935 K5
      PLS     M926  ; #8 -> #7
2209  LD      M924  ; #6 -> #5
      BMOV    D935 D930 K5
      PLS     M925  ; #7 -> #6
2216  LD      M923  ; #5 -> #4
      BMOV    D930 D925 K5
      PLS     M924  ; #6 -> #5
2223  LD      M922  ; #4 -> #3
      BMOV    D925 D920 K5
      PLS     M923  ; #5 -> #4
2230  LD      M921  ; #3 -> #2
      BMOV    D920 D915 K5
      PLS     M922  ; #4 -> #3
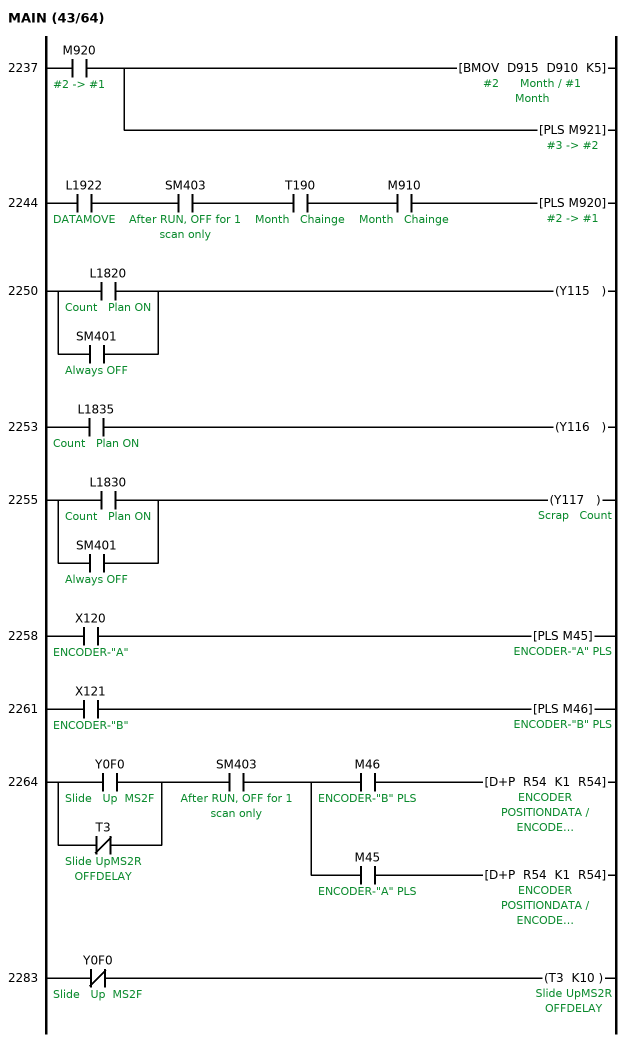
2237  LD      M920  ; #2 -> #1
      BMOV    D915 D910 K5
      PLS     M921  ; #3 -> #2
2244  LD      L1922  ; DATAMOVE
      AND     SM403  ; After RUN, OFF for 1 scan only
      AND     T190  ; Month   Chainge
      AND     M910  ; Month   Chainge
      PLS     M920  ; #2 -> #1
2250  LD      L1820  ; Count   Plan ON
      OR      SM401  ; Always OFF
      OUT     Y115
2253  LD      L1835  ; Count   Plan ON
      OUT     Y116
2255  LD      L1830  ; Count   Plan ON
      OR      SM401  ; Always OFF
      OUT     Y117  ; Scrap   Count
2258  LD      X120  ; ENCODER-"A"
      PLS     M45  ; ENCODER-"A" PLS
2261  LD      X121  ; ENCODER-"B"
      PLS     M46  ; ENCODER-"B" PLS
2264  LD      Y0F0  ; Slide   Up  MS2F
      ORI     T3  ; Slide UpMS2R OFFDELAY
      AND     SM403  ; After RUN, OFF for 1 scan only
      MPS
      AND     M46  ; ENCODER-"B" PLS
      D+P     R54 K1 R54  ; ENCODER POSITIONDATA
      MPP
      AND     M45  ; ENCODER-"A" PLS
      D+P     R54 K1 R54
2283  LDI     Y0F0  ; Slide   Up  MS2F
      OUT     T3 K10  ; Slide UpMS2R OFFDELAY
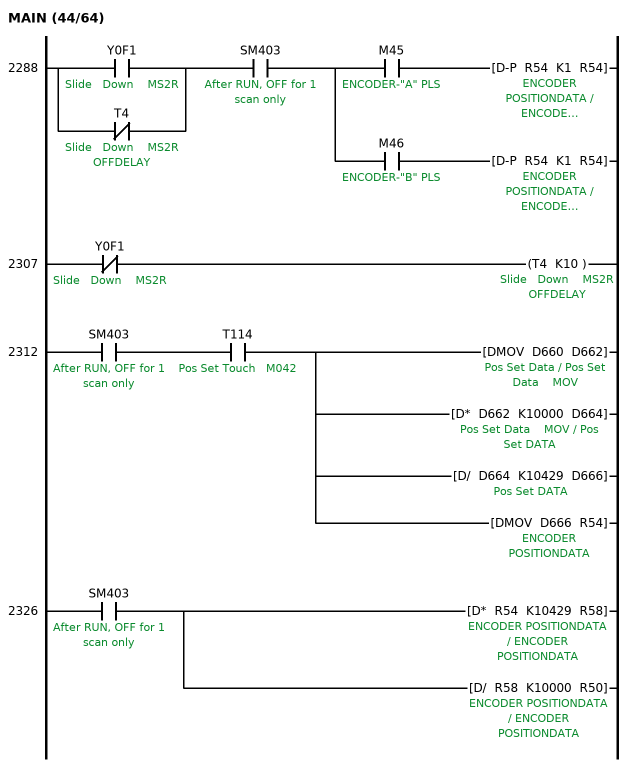
2288  LD      Y0F1  ; Slide   Down    MS2R
      ORI     T4  ; Slide   Down    MS2R OFFDELAY
      AND     SM403  ; After RUN, OFF for 1 scan only
      MPS
      AND     M45  ; ENCODER-"A" PLS
      D-P     R54 K1 R54
      MPP
      AND     M46  ; ENCODER-"B" PLS
      D-P     R54 K1 R54
2307  LDI     Y0F1  ; Slide   Down    MS2R
      OUT     T4 K10  ; Slide   Down    MS2R OFFDELAY
2312  LD      SM403  ; After RUN, OFF for 1 scan only
      AND     T114  ; Pos Set Touch   M042
      DMOV    D660 D662  ; Pos Set Data / Pos Set Data    MOV
      D*      D662 K10000 D664  ; Pos Set DATA
      D/      D664 K10429 D666
      DMOV    D666 R54
2326  LD      SM403  ; After RUN, OFF for 1 scan only
      D*      R54 K10429 R58  ; ENCODER POSITIONDATA
      D/      R58 K10000 R50  ; ENCODER POSITIONDATA
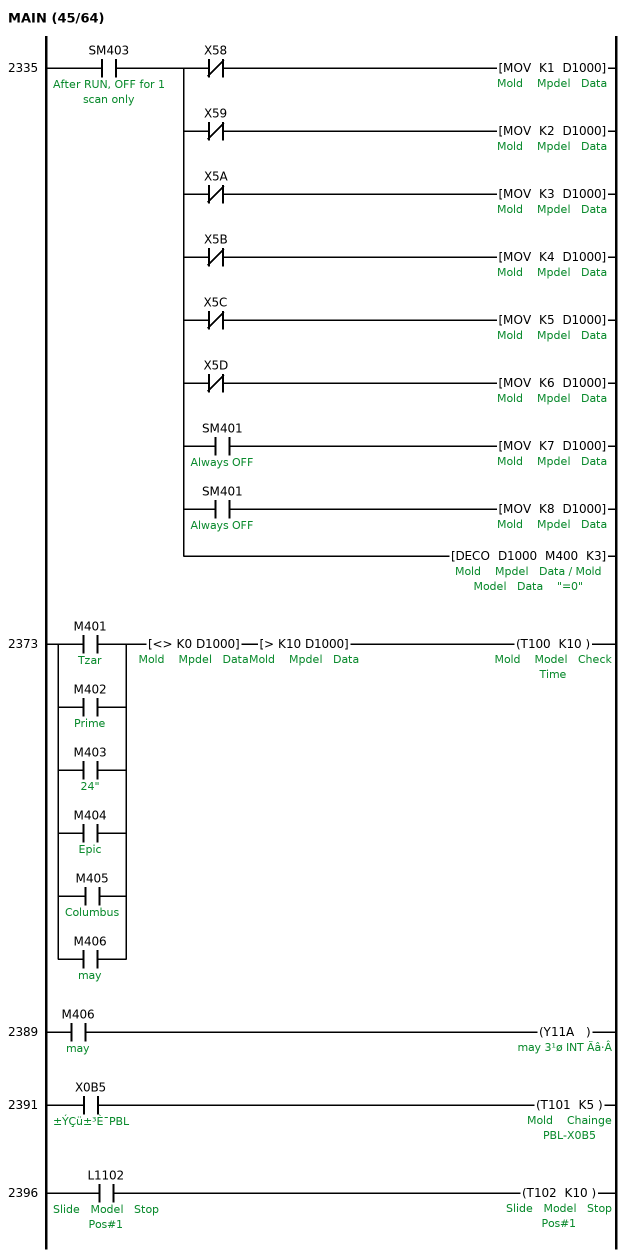
2335  LD      SM403  ; After RUN, OFF for 1 scan only
      MPS
      ANI     X58
      MOV     K1 D1000  ; Mold    Mpdel   Data
      MRD
      ANI     X59
      MOV     K2 D1000
      MRD
      ANI     X5A
      MOV     K3 D1000
      MRD
      ANI     X5B
      MOV     K4 D1000
      MRD
      ANI     X5C
      MOV     K5 D1000
      MRD
      ANI     X5D
      MOV     K6 D1000
      MRD
      AND     SM401  ; Always OFF
      MOV     K7 D1000
      MRD
      AND     SM401  ; Always OFF
      MOV     K8 D1000
      MPP
      DECO    D1000 M400 K3  ; Mold    Model   Data    "=0"
2373  LD      M401  ; Tzar
      OR      M402  ; Prime
      OR      M403  ; 24"
      OR      M404  ; Epic
      OR      M405  ; Columbus
      OR      M406  ; may
      AND<>   K0 D1000  ; Mold    Mpdel   Data
      AND>    K10 D1000  ; Mold    Mpdel   Data
      OUT     T100 K10  ; Mold    Model   Check   Time
2389  LD      M406  ; may
      OUT     Y11A  ; may 3¹ø INT Ãâ·Â
2391  LD      X0B5  ; ±ÝÇü±³È¯PBL
      OUT     T101 K5  ; Mold    Chainge PBL-X0B5
2396  LD      L1102  ; Slide   Model   Stop    Pos#1
      OUT     T102 K10  ; Slide   Model   Stop    Pos#1
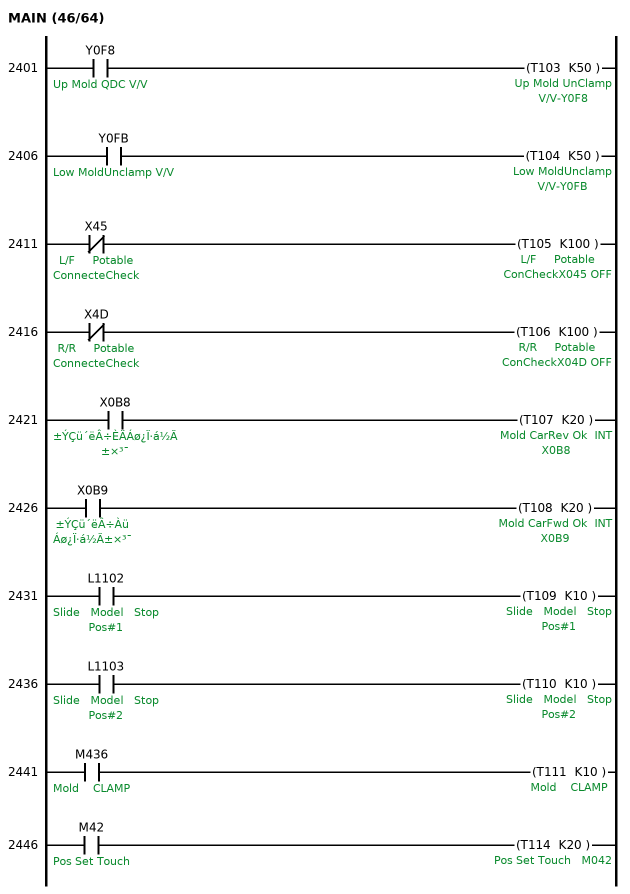
2401  LD      Y0F8  ; Up Mold QDC V/V
      OUT     T103 K50  ; Up Mold UnClamp V/V-Y0F8
2406  LD      Y0FB  ; Low MoldUnclamp V/V
      OUT     T104 K50  ; Low MoldUnclamp V/V-Y0FB
2411  LDI     X45  ; L/F     Potable ConnecteCheck
      OUT     T105 K100  ; L/F     Potable ConCheckX045 OFF
2416  LDI     X4D  ; R/R     Potable ConnecteCheck
      OUT     T106 K100  ; R/R     Potable ConCheckX04D OFF
2421  LD      X0B8  ; ±ÝÇü´ëÂ÷ÈÄÁø¿Ï·á½Ã±×³¯
      OUT     T107 K20  ; Mold CarRev Ok  INT X0B8
2426  LD      X0B9  ; ±ÝÇü´ëÂ÷ÀüÁø¿Ï·á½Ã±×³¯
      OUT     T108 K20  ; Mold CarFwd Ok  INT X0B9
2431  LD      L1102  ; Slide   Model   Stop    Pos#1
      OUT     T109 K10  ; Slide   Model   Stop    Pos#1
2436  LD      L1103  ; Slide   Model   Stop    Pos#2
      OUT     T110 K10  ; Slide   Model   Stop    Pos#2
2441  LD      M436  ; Mold    CLAMP
      OUT     T111 K10  ; Mold    CLAMP
2446  LD      M42  ; Pos Set Touch
      OUT     T114 K20  ; Pos Set Touch   M042
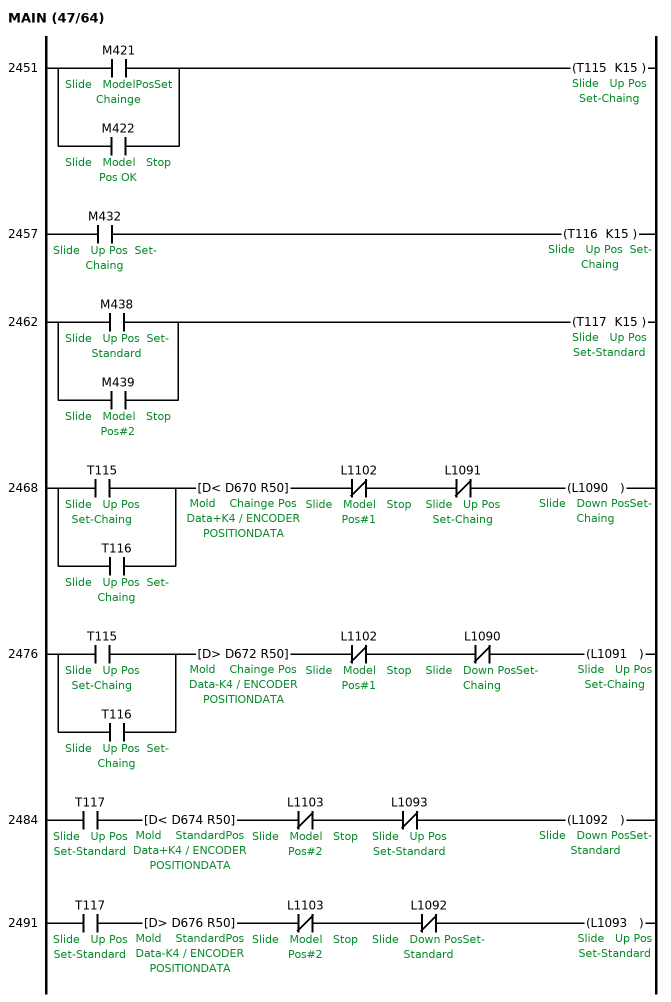
2451  LD      M421  ; Slide   ModelPosSet     Chainge
      OR      M422  ; Slide   Model   Stop    Pos OK
      OUT     T115 K15  ; Slide   Up Pos  Set-Chaing
2457  LD      M432  ; Slide   Up Pos  Set-    Chaing
      OUT     T116 K15  ; Slide   Up Pos  Set-    Chaing
2462  LD      M438  ; Slide   Up Pos  Set-    Standard
      OR      M439  ; Slide   Model   Stop    Pos#2
      OUT     T117 K15  ; Slide   Up Pos  Set-Standard
2468  LD      T115  ; Slide   Up Pos  Set-Chaing
      OR      T116  ; Slide   Up Pos  Set-    Chaing
      ANDD<   D670 R50  ; Mold    Chainge Pos Data+K4 / ENCODER POSITIONDATA
      ANI     L1102  ; Slide   Model   Stop    Pos#1
      ANI     L1091  ; Slide   Up Pos  Set-Chaing
      OUT     L1090  ; Slide   Down PosSet-    Chaing
2476  LD      T115  ; Slide   Up Pos  Set-Chaing
      OR      T116  ; Slide   Up Pos  Set-    Chaing
      ANDD>   D672 R50  ; Mold    Chainge Pos Data-K4 / ENCODER POSITIONDATA
      ANI     L1102  ; Slide   Model   Stop    Pos#1
      ANI     L1090  ; Slide   Down PosSet-    Chaing
      OUT     L1091  ; Slide   Up Pos  Set-Chaing
2484  LD      T117  ; Slide   Up Pos  Set-Standard
      ANDD<   D674 R50  ; Mold    StandardPos Data+K4 / ENCODER POSITIONDATA
      ANI     L1103  ; Slide   Model   Stop    Pos#2
      ANI     L1093  ; Slide   Up Pos  Set-Standard
      OUT     L1092  ; Slide   Down PosSet-    Standard
2491  LD      T117  ; Slide   Up Pos  Set-Standard
      ANDD>   D676 R50  ; Mold    StandardPos Data-K4 / ENCODER POSITIONDATA
      ANI     L1103  ; Slide   Model   Stop    Pos#2
      ANI     L1092  ; Slide   Down PosSet-    Standard
      OUT     L1093  ; Slide   Up Pos  Set-Standard
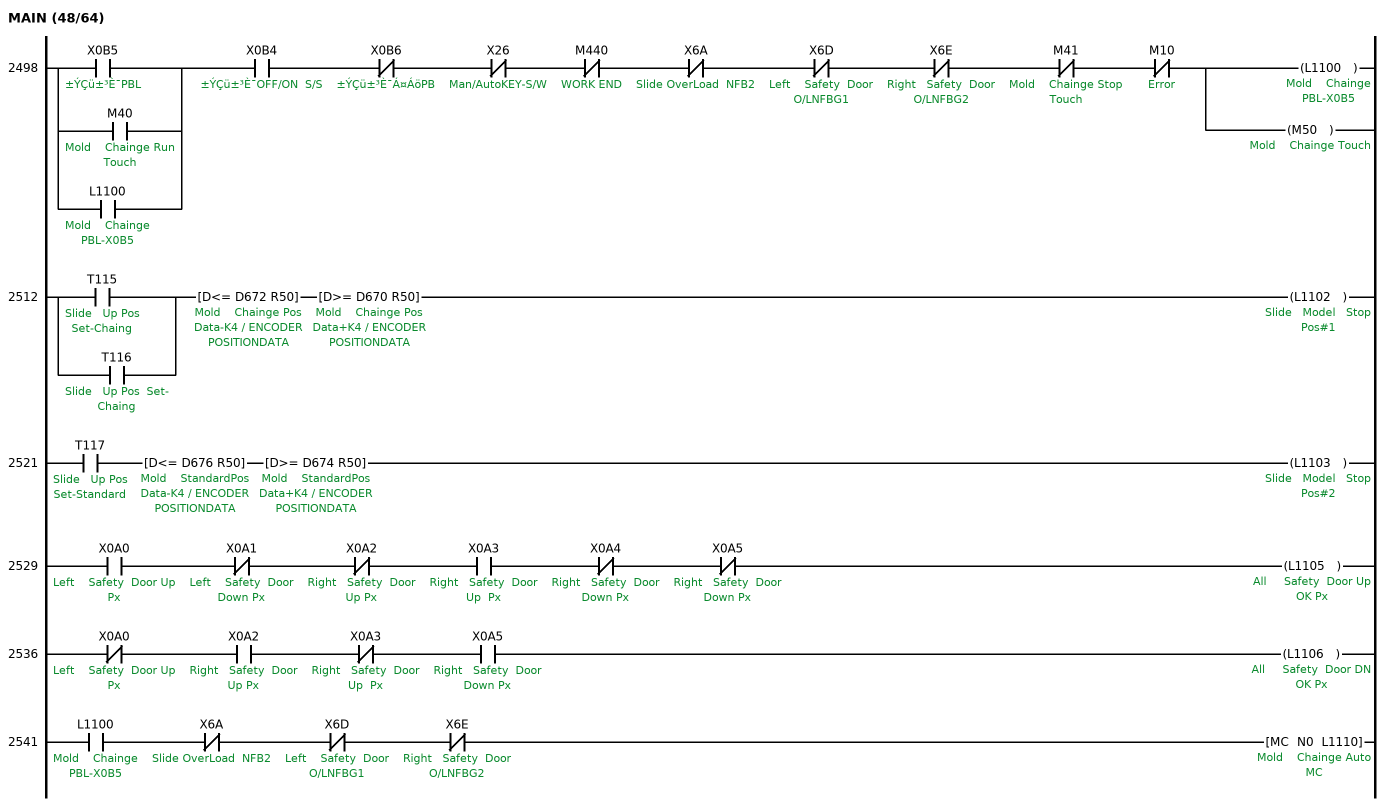
2498  LD      X0B5  ; ±ÝÇü±³È¯PBL
      OR      M40  ; Mold    Chainge Run     Touch
      OR      L1100  ; Mold    Chainge PBL-X0B5
      AND     X0B4  ; ±ÝÇü±³È¯OFF/ON  S/S
      ANI     X0B6  ; ±ÝÇü±³È¯Á¤ÁöPB
      ANI     X26  ; Man/AutoKEY-S/W
      ANI     M440  ; WORK END
      ANI     X6A  ; Slide OverLoad  NFB2
      ANI     X6D  ; Left    Safety  Door O/LNFBG1
      ANI     X6E  ; Right   Safety  Door O/LNFBG2
      ANI     M41  ; Mold    Chainge Stop    Touch
      ANI     M10  ; Error
      OUT     L1100  ; Mold    Chainge PBL-X0B5
      OUT     M50  ; Mold    Chainge Touch
2512  LD      T115  ; Slide   Up Pos  Set-Chaing
      OR      T116  ; Slide   Up Pos  Set-    Chaing
      ANDD<=  D672 R50  ; Mold    Chainge Pos Data-K4 / ENCODER POSITIONDATA
      ANDD>=  D670 R50  ; Mold    Chainge Pos Data+K4 / ENCODER POSITIONDATA
      OUT     L1102  ; Slide   Model   Stop    Pos#1
2521  LD      T117  ; Slide   Up Pos  Set-Standard
      ANDD<=  D676 R50  ; Mold    StandardPos Data-K4 / ENCODER POSITIONDATA
      ANDD>=  D674 R50  ; Mold    StandardPos Data+K4 / ENCODER POSITIONDATA
      OUT     L1103  ; Slide   Model   Stop    Pos#2
2529  LD      X0A0  ; Left    Safety  Door Up Px
      ANI     X0A1  ; Left    Safety  Door    Down Px
      ANI     X0A2  ; Right   Safety  Door Up Px
      AND     X0A3  ; Right   Safety  Door Up  Px
      ANI     X0A4  ; Right   Safety  Door    Down Px
      ANI     X0A5  ; Right   Safety  Door    Down Px
      OUT     L1105  ; All     Safety  Door Up OK Px
2536  LDI     X0A0  ; Left    Safety  Door Up Px
      AND     X0A2  ; Right   Safety  Door Up Px
      ANI     X0A3  ; Right   Safety  Door Up  Px
      AND     X0A5  ; Right   Safety  Door    Down Px
      OUT     L1106  ; All     Safety  Door DN OK Px
2541  LD      L1100  ; Mold    Chainge PBL-X0B5
      ANI     X6A  ; Slide OverLoad  NFB2
      ANI     X6D  ; Left    Safety  Door O/LNFBG1
      ANI     X6E  ; Right   Safety  Door O/LNFBG2
      MC      N0 L1110
